//{attribute 'qualified_only'}
VAR_GLOBAL
    {attribute 'pytmc' := '
        pv: PLC:LAMP:VAC:OVRDON
        io: io
    '}
    xSystemOverrideMode_LAMP	: BOOL := FALSE; (* Global system override for the HXR Vacuum System EBD*)

    {attribute 'pytmc' := '
        pv: PLC:LAMP:ON:BEAMLINE
        io:io
    '}
    xOnBeamline	:	BOOL := TRUE; (*Always assume On Beamline for safety checks*)

    rHighVoltageMinPressure	: REAL := 1e-05; (*Hard coded High voltage Minimum Enable Pressure*)

END_VAR

(* stored: Version 1.1.0.1, ProductVersion 3.1.4022.18
   GVL GVL_Variables: Id {c498846d-d5de-49b1-923d-af8c367da0a5} *)
